Omron CX-Programmer project NewProject (CX-Programmer 9.73)

# PLC NewPLC1: CP1E N20

## Global symbols (name address type ; comment)
0.00 BOOL  ; PB START
0.02 BOOL  ; PB STOP
100.01 BOOL  ; LED 1
100.02 BOOL  ; LED 2
100.03 BOOL  ; LED 3
100.04 BOOL  ; LED 4
200.01 BOOL  ; RELAY
T001 BOOL  ; TIMER 1
T002 BOOL  ; TIMER 2
T003 BOOL  ; TIMER 3

## Program NewProgram1 (cyclic task 0)

### Section Section1

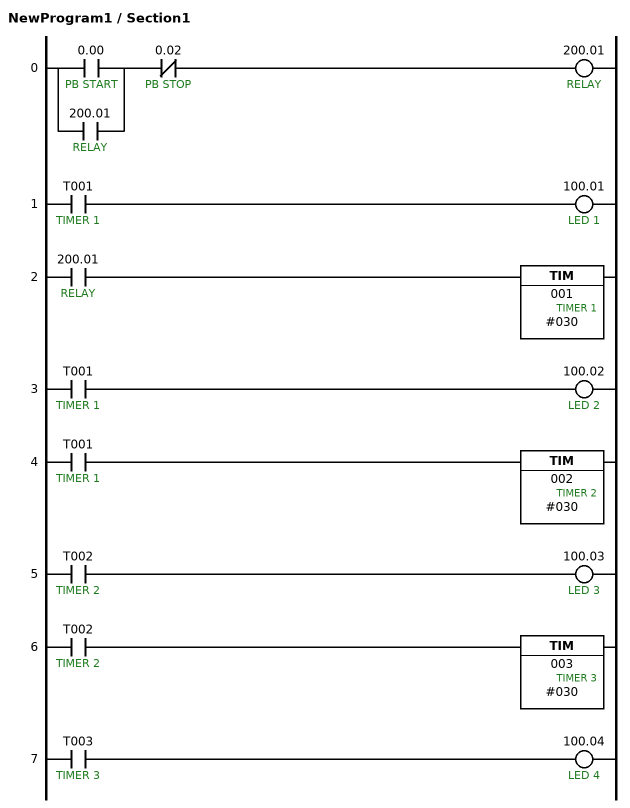
; rung 0
LD 0.00  ; PB START
OR 200.01  ; RELAY
ANDNOT 0.02  ; PB STOP
OUT 200.01  ; RELAY
; rung 1
LD T001  ; TIMER 1
OUT 100.01  ; LED 1
; rung 2
LD 200.01  ; RELAY
TIM 001 #030  ; TIMER 1
; rung 3
LD T001  ; TIMER 1
OUT 100.02  ; LED 2
; rung 4
LD T001  ; TIMER 1
TIM 002 #030  ; TIMER 2
; rung 5
LD T002  ; TIMER 2
OUT 100.03  ; LED 3
; rung 6
LD T002  ; TIMER 2
TIM 003 #030  ; TIMER 3
; rung 7
LD T003  ; TIMER 3
OUT 100.04  ; LED 4

### Section END
; rung 0
END(001)